# EPICS autosave request: support/ip/2-9/ipApp/Db/Newport_LAE500_settings.req
$(P)$(R)_READ_DATA.SCAN
$(P)$(R)_READ_STATUS.SCAN
$(P)$(R)_REMOTE.VAL
$(P)$(R)_Y_COEFF.VAL
$(P)$(R)_Z_COEFF.VAL
$(P)$(R)_INTEGRATE.VAL
$(P)$(R)_INCREMENT.VAL
$(P)$(R)_UNITS.VAL
